// TIA Portal V20 export
ORGANIZATION_BLOCK "Main"   // OB1, LAD, ProgramCycle
TITLE = "Main Program Sweep (Cycle)"
{ S7_Optimized_Access := 'TRUE' }
// stored: SetENOAutomatically false
   VAR_INPUT
      Initial_Call : Bool;   // Initial call of this OB
      Remanence : Bool;   // =True, if remanent data are available
   END_VAR
BEGIN

REGION Network 1
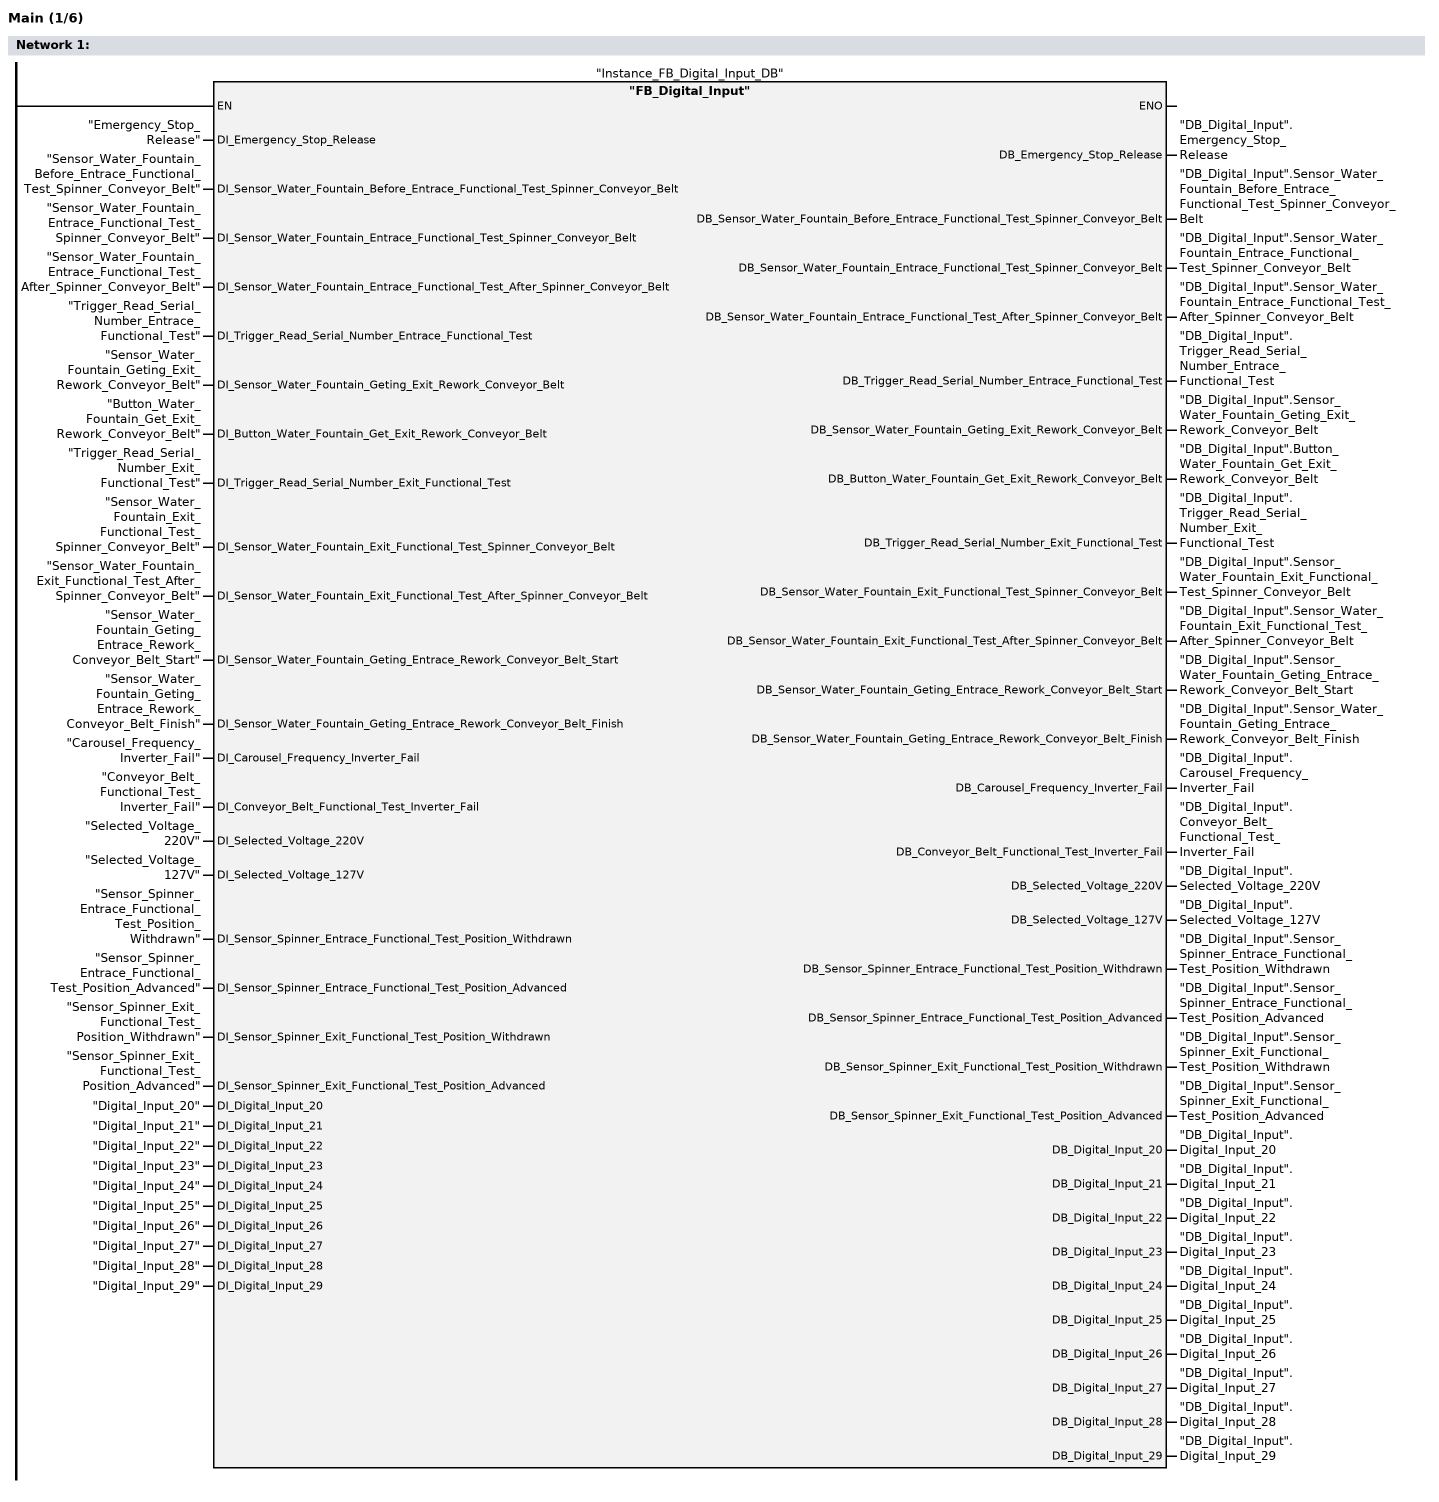
   RUNG wire#powerrail
      "Instance_FB_Digital_Input_DB"(DI_Emergency_Stop_Release := "Emergency_Stop_Release", DI_Sensor_Water_Fountain_Before_Entrace_Functional_Test_Spinner_Conveyor_Belt := "Sensor_Water_Fountain_Before_Entrace_Functional_Test_Spinner_Conveyor_Belt", DI_Sensor_Water_Fountain_Entrace_Functional_Test_Spinner_Conveyor_Belt := "Sensor_Water_Fountain_Entrace_Functional_Test_Spinner_Conveyor_Belt", DI_Sensor_Water_Fountain_Entrace_Functional_Test_After_Spinner_Conveyor_Belt := "Sensor_Water_Fountain_Entrace_Functional_Test_After_Spinner_Conveyor_Belt", DI_Trigger_Read_Serial_Number_Entrace_Functional_Test := "Trigger_Read_Serial_Number_Entrace_Functional_Test", DI_Sensor_Water_Fountain_Geting_Exit_Rework_Conveyor_Belt := "Sensor_Water_Fountain_Geting_Exit_Rework_Conveyor_Belt", DI_Button_Water_Fountain_Get_Exit_Rework_Conveyor_Belt := "Button_Water_Fountain_Get_Exit_Rework_Conveyor_Belt", DI_Trigger_Read_Serial_Number_Exit_Functional_Test := "Trigger_Read_Serial_Number_Exit_Functional_Test", DI_Sensor_Water_Fountain_Exit_Functional_Test_Spinner_Conveyor_Belt := "Sensor_Water_Fountain_Exit_Functional_Test_Spinner_Conveyor_Belt", DI_Sensor_Water_Fountain_Exit_Functional_Test_After_Spinner_Conveyor_Belt := "Sensor_Water_Fountain_Exit_Functional_Test_After_Spinner_Conveyor_Belt", DI_Sensor_Water_Fountain_Geting_Entrace_Rework_Conveyor_Belt_Start := "Sensor_Water_Fountain_Geting_Entrace_Rework_Conveyor_Belt_Start", DI_Sensor_Water_Fountain_Geting_Entrace_Rework_Conveyor_Belt_Finish := "Sensor_Water_Fountain_Geting_Entrace_Rework_Conveyor_Belt_Finish", DI_Carousel_Frequency_Inverter_Fail := "Carousel_Frequency_Inverter_Fail", DI_Conveyor_Belt_Functional_Test_Inverter_Fail := "Conveyor_Belt_Functional_Test_Inverter_Fail", DI_Selected_Voltage_220V := "Selected_Voltage_220V", DI_Selected_Voltage_127V := "Selected_Voltage_127V", DI_Sensor_Spinner_Entrace_Functional_Test_Position_Withdrawn := "Sensor_Spinner_Entrace_Functional_Test_Position_Withdrawn", DI_Sensor_Spinner_Entrace_Functional_Test_Position_Advanced := "Sensor_Spinner_Entrace_Functional_Test_Position_Advanced", DI_Sensor_Spinner_Exit_Functional_Test_Position_Withdrawn := "Sensor_Spinner_Exit_Functional_Test_Position_Withdrawn", DI_Sensor_Spinner_Exit_Functional_Test_Position_Advanced := "Sensor_Spinner_Exit_Functional_Test_Position_Advanced", DI_Digital_Input_20 := "Digital_Input_20", DI_Digital_Input_21 := "Digital_Input_21", DI_Digital_Input_22 := "Digital_Input_22", DI_Digital_Input_23 := "Digital_Input_23", DI_Digital_Input_24 := "Digital_Input_24", DI_Digital_Input_25 := "Digital_Input_25", DI_Digital_Input_26 := "Digital_Input_26", DI_Digital_Input_27 := "Digital_Input_27", DI_Digital_Input_28 := "Digital_Input_28", DI_Digital_Input_29 := "Digital_Input_29", DB_Emergency_Stop_Release => "DB_Digital_Input".Emergency_Stop_Release, DB_Sensor_Water_Fountain_Before_Entrace_Functional_Test_Spinner_Conveyor_Belt => "DB_Digital_Input".Sensor_Water_Fountain_Before_Entrace_Functional_Test_Spinner_Conveyor_Belt, DB_Sensor_Water_Fountain_Entrace_Functional_Test_Spinner_Conveyor_Belt => "DB_Digital_Input".Sensor_Water_Fountain_Entrace_Functional_Test_Spinner_Conveyor_Belt, DB_Sensor_Water_Fountain_Entrace_Functional_Test_After_Spinner_Conveyor_Belt => "DB_Digital_Input".Sensor_Water_Fountain_Entrace_Functional_Test_After_Spinner_Conveyor_Belt, DB_Trigger_Read_Serial_Number_Entrace_Functional_Test => "DB_Digital_Input".Trigger_Read_Serial_Number_Entrace_Functional_Test, DB_Sensor_Water_Fountain_Geting_Exit_Rework_Conveyor_Belt => "DB_Digital_Input".Sensor_Water_Fountain_Geting_Exit_Rework_Conveyor_Belt, DB_Button_Water_Fountain_Get_Exit_Rework_Conveyor_Belt => "DB_Digital_Input".Button_Water_Fountain_Get_Exit_Rework_Conveyor_Belt, DB_Trigger_Read_Serial_Number_Exit_Functional_Test => "DB_Digital_Input".Trigger_Read_Serial_Number_Exit_Functional_Test, DB_Sensor_Water_Fountain_Exit_Functional_Test_Spinner_Conveyor_Belt => "DB_Digital_Input".Sensor_Water_Fountain_Exit_Functional_Test_Spinner_Conveyor_Belt, DB_Sensor_Water_Fountain_Exit_Functional_Test_After_Spinner_Conveyor_Belt => "DB_Digital_Input".Sensor_Water_Fountain_Exit_Functional_Test_After_Spinner_Conveyor_Belt, DB_Sensor_Water_Fountain_Geting_Entrace_Rework_Conveyor_Belt_Start => "DB_Digital_Input".Sensor_Water_Fountain_Geting_Entrace_Rework_Conveyor_Belt_Start, DB_Sensor_Water_Fountain_Geting_Entrace_Rework_Conveyor_Belt_Finish => "DB_Digital_Input".Sensor_Water_Fountain_Geting_Entrace_Rework_Conveyor_Belt_Finish, DB_Carousel_Frequency_Inverter_Fail => "DB_Digital_Input".Carousel_Frequency_Inverter_Fail, DB_Conveyor_Belt_Functional_Test_Inverter_Fail => "DB_Digital_Input".Conveyor_Belt_Functional_Test_Inverter_Fail, DB_Selected_Voltage_220V => "DB_Digital_Input".Selected_Voltage_220V, DB_Selected_Voltage_127V => "DB_Digital_Input".Selected_Voltage_127V, DB_Sensor_Spinner_Entrace_Functional_Test_Position_Withdrawn => "DB_Digital_Input".Sensor_Spinner_Entrace_Functional_Test_Position_Withdrawn, DB_Sensor_Spinner_Entrace_Functional_Test_Position_Advanced => "DB_Digital_Input".Sensor_Spinner_Entrace_Functional_Test_Position_Advanced, DB_Sensor_Spinner_Exit_Functional_Test_Position_Withdrawn => "DB_Digital_Input".Sensor_Spinner_Exit_Functional_Test_Position_Withdrawn, DB_Sensor_Spinner_Exit_Functional_Test_Position_Advanced => "DB_Digital_Input".Sensor_Spinner_Exit_Functional_Test_Position_Advanced, DB_Digital_Input_20 => "DB_Digital_Input".Digital_Input_20, DB_Digital_Input_21 => "DB_Digital_Input".Digital_Input_21, DB_Digital_Input_22 => "DB_Digital_Input".Digital_Input_22, DB_Digital_Input_23 => "DB_Digital_Input".Digital_Input_23, DB_Digital_Input_24 => "DB_Digital_Input".Digital_Input_24, DB_Digital_Input_25 => "DB_Digital_Input".Digital_Input_25, DB_Digital_Input_26 => "DB_Digital_Input".Digital_Input_26, DB_Digital_Input_27 => "DB_Digital_Input".Digital_Input_27, DB_Digital_Input_28 => "DB_Digital_Input".Digital_Input_28, DB_Digital_Input_29 => "DB_Digital_Input".Digital_Input_29)
   END_RUNG
   // the same network as SCL:
   "Instance_FB_Digital_Input_DB"(DI_Emergency_Stop_Release := "Emergency_Stop_Release",   // "FB_Digital_Input"
                           DI_Sensor_Water_Fountain_Before_Entrace_Functional_Test_Spinner_Conveyor_Belt := "Sensor_Water_Fountain_Before_Entrace_Functional_Test_Spinner_Conveyor_Belt",
                           DI_Sensor_Water_Fountain_Entrace_Functional_Test_Spinner_Conveyor_Belt := "Sensor_Water_Fountain_Entrace_Functional_Test_Spinner_Conveyor_Belt",
                           DI_Sensor_Water_Fountain_Entrace_Functional_Test_After_Spinner_Conveyor_Belt := "Sensor_Water_Fountain_Entrace_Functional_Test_After_Spinner_Conveyor_Belt",
                           DI_Trigger_Read_Serial_Number_Entrace_Functional_Test := "Trigger_Read_Serial_Number_Entrace_Functional_Test",
                           DI_Sensor_Water_Fountain_Geting_Exit_Rework_Conveyor_Belt := "Sensor_Water_Fountain_Geting_Exit_Rework_Conveyor_Belt",
                           DI_Button_Water_Fountain_Get_Exit_Rework_Conveyor_Belt := "Button_Water_Fountain_Get_Exit_Rework_Conveyor_Belt",
                           DI_Trigger_Read_Serial_Number_Exit_Functional_Test := "Trigger_Read_Serial_Number_Exit_Functional_Test",
                           DI_Sensor_Water_Fountain_Exit_Functional_Test_Spinner_Conveyor_Belt := "Sensor_Water_Fountain_Exit_Functional_Test_Spinner_Conveyor_Belt",
                           DI_Sensor_Water_Fountain_Exit_Functional_Test_After_Spinner_Conveyor_Belt := "Sensor_Water_Fountain_Exit_Functional_Test_After_Spinner_Conveyor_Belt",
                           DI_Sensor_Water_Fountain_Geting_Entrace_Rework_Conveyor_Belt_Start := "Sensor_Water_Fountain_Geting_Entrace_Rework_Conveyor_Belt_Start",
                           DI_Sensor_Water_Fountain_Geting_Entrace_Rework_Conveyor_Belt_Finish := "Sensor_Water_Fountain_Geting_Entrace_Rework_Conveyor_Belt_Finish",
                           DI_Carousel_Frequency_Inverter_Fail := "Carousel_Frequency_Inverter_Fail",
                           DI_Conveyor_Belt_Functional_Test_Inverter_Fail := "Conveyor_Belt_Functional_Test_Inverter_Fail",
                           DI_Selected_Voltage_220V := "Selected_Voltage_220V",
                           DI_Selected_Voltage_127V := "Selected_Voltage_127V",
                           DI_Sensor_Spinner_Entrace_Functional_Test_Position_Withdrawn := "Sensor_Spinner_Entrace_Functional_Test_Position_Withdrawn",
                           DI_Sensor_Spinner_Entrace_Functional_Test_Position_Advanced := "Sensor_Spinner_Entrace_Functional_Test_Position_Advanced",
                           DI_Sensor_Spinner_Exit_Functional_Test_Position_Withdrawn := "Sensor_Spinner_Exit_Functional_Test_Position_Withdrawn",
                           DI_Sensor_Spinner_Exit_Functional_Test_Position_Advanced := "Sensor_Spinner_Exit_Functional_Test_Position_Advanced",
                           DI_Digital_Input_20 := "Digital_Input_20",
                           DI_Digital_Input_21 := "Digital_Input_21",
                           DI_Digital_Input_22 := "Digital_Input_22",
                           DI_Digital_Input_23 := "Digital_Input_23",
                           DI_Digital_Input_24 := "Digital_Input_24",
                           DI_Digital_Input_25 := "Digital_Input_25",
                           DI_Digital_Input_26 := "Digital_Input_26",
                           DI_Digital_Input_27 := "Digital_Input_27",
                           DI_Digital_Input_28 := "Digital_Input_28",
                           DI_Digital_Input_29 := "Digital_Input_29",
                           DB_Emergency_Stop_Release => "DB_Digital_Input".Emergency_Stop_Release,
                           DB_Sensor_Water_Fountain_Before_Entrace_Functional_Test_Spinner_Conveyor_Belt => "DB_Digital_Input".Sensor_Water_Fountain_Before_Entrace_Functional_Test_Spinner_Conveyor_Belt,
                           DB_Sensor_Water_Fountain_Entrace_Functional_Test_Spinner_Conveyor_Belt => "DB_Digital_Input".Sensor_Water_Fountain_Entrace_Functional_Test_Spinner_Conveyor_Belt,
                           DB_Sensor_Water_Fountain_Entrace_Functional_Test_After_Spinner_Conveyor_Belt => "DB_Digital_Input".Sensor_Water_Fountain_Entrace_Functional_Test_After_Spinner_Conveyor_Belt,
                           DB_Trigger_Read_Serial_Number_Entrace_Functional_Test => "DB_Digital_Input".Trigger_Read_Serial_Number_Entrace_Functional_Test,
                           DB_Sensor_Water_Fountain_Geting_Exit_Rework_Conveyor_Belt => "DB_Digital_Input".Sensor_Water_Fountain_Geting_Exit_Rework_Conveyor_Belt,
                           DB_Button_Water_Fountain_Get_Exit_Rework_Conveyor_Belt => "DB_Digital_Input".Button_Water_Fountain_Get_Exit_Rework_Conveyor_Belt,
                           DB_Trigger_Read_Serial_Number_Exit_Functional_Test => "DB_Digital_Input".Trigger_Read_Serial_Number_Exit_Functional_Test,
                           DB_Sensor_Water_Fountain_Exit_Functional_Test_Spinner_Conveyor_Belt => "DB_Digital_Input".Sensor_Water_Fountain_Exit_Functional_Test_Spinner_Conveyor_Belt,
                           DB_Sensor_Water_Fountain_Exit_Functional_Test_After_Spinner_Conveyor_Belt => "DB_Digital_Input".Sensor_Water_Fountain_Exit_Functional_Test_After_Spinner_Conveyor_Belt,
                           DB_Sensor_Water_Fountain_Geting_Entrace_Rework_Conveyor_Belt_Start => "DB_Digital_Input".Sensor_Water_Fountain_Geting_Entrace_Rework_Conveyor_Belt_Start,
                           DB_Sensor_Water_Fountain_Geting_Entrace_Rework_Conveyor_Belt_Finish => "DB_Digital_Input".Sensor_Water_Fountain_Geting_Entrace_Rework_Conveyor_Belt_Finish,
                           DB_Carousel_Frequency_Inverter_Fail => "DB_Digital_Input".Carousel_Frequency_Inverter_Fail,
                           DB_Conveyor_Belt_Functional_Test_Inverter_Fail => "DB_Digital_Input".Conveyor_Belt_Functional_Test_Inverter_Fail,
                           DB_Selected_Voltage_220V => "DB_Digital_Input".Selected_Voltage_220V,
                           DB_Selected_Voltage_127V => "DB_Digital_Input".Selected_Voltage_127V,
                           DB_Sensor_Spinner_Entrace_Functional_Test_Position_Withdrawn => "DB_Digital_Input".Sensor_Spinner_Entrace_Functional_Test_Position_Withdrawn,
                           DB_Sensor_Spinner_Entrace_Functional_Test_Position_Advanced => "DB_Digital_Input".Sensor_Spinner_Entrace_Functional_Test_Position_Advanced,
                           DB_Sensor_Spinner_Exit_Functional_Test_Position_Withdrawn => "DB_Digital_Input".Sensor_Spinner_Exit_Functional_Test_Position_Withdrawn,
                           DB_Sensor_Spinner_Exit_Functional_Test_Position_Advanced => "DB_Digital_Input".Sensor_Spinner_Exit_Functional_Test_Position_Advanced,
                           DB_Digital_Input_20 => "DB_Digital_Input".Digital_Input_20,
                           DB_Digital_Input_21 => "DB_Digital_Input".Digital_Input_21,
                           DB_Digital_Input_22 => "DB_Digital_Input".Digital_Input_22,
                           DB_Digital_Input_23 => "DB_Digital_Input".Digital_Input_23,
                           DB_Digital_Input_24 => "DB_Digital_Input".Digital_Input_24,
                           DB_Digital_Input_25 => "DB_Digital_Input".Digital_Input_25,
                           DB_Digital_Input_26 => "DB_Digital_Input".Digital_Input_26,
                           DB_Digital_Input_27 => "DB_Digital_Input".Digital_Input_27,
                           DB_Digital_Input_28 => "DB_Digital_Input".Digital_Input_28,
                           DB_Digital_Input_29 => "DB_Digital_Input".Digital_Input_29);
END_REGION

REGION Network 2
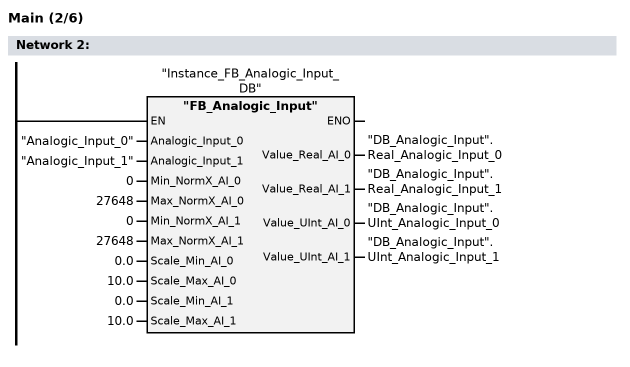
   RUNG wire#powerrail
      "Instance_FB_Analogic_Input_DB"(Analogic_Input_0 := "Analogic_Input_0", Analogic_Input_1 := "Analogic_Input_1", Min_NormX_AI_0 := 0, Max_NormX_AI_0 := 27648, Min_NormX_AI_1 := 0, Max_NormX_AI_1 := 27648, Scale_Min_AI_0 := 0.0, Scale_Max_AI_0 := 10.0, Scale_Min_AI_1 := 0.0, Scale_Max_AI_1 := 10.0, Value_Real_AI_0 => "DB_Analogic_Input".Real_Analogic_Input_0, Value_Real_AI_1 => "DB_Analogic_Input".Real_Analogic_Input_1, Value_UInt_AI_0 => "DB_Analogic_Input".UInt_Analogic_Input_0, Value_UInt_AI_1 => "DB_Analogic_Input".UInt_Analogic_Input_1)
   END_RUNG
   // the same network as SCL:
   "Instance_FB_Analogic_Input_DB"(Analogic_Input_0 := "Analogic_Input_0",   // "FB_Analogic_Input"
                           Analogic_Input_1 := "Analogic_Input_1",
                           Min_NormX_AI_0 := 0,
                           Max_NormX_AI_0 := 27648,
                           Min_NormX_AI_1 := 0,
                           Max_NormX_AI_1 := 27648,
                           Scale_Min_AI_0 := 0.0,
                           Scale_Max_AI_0 := 10.0,
                           Scale_Min_AI_1 := 0.0,
                           Scale_Max_AI_1 := 10.0,
                           Value_Real_AI_0 => "DB_Analogic_Input".Real_Analogic_Input_0,
                           Value_Real_AI_1 => "DB_Analogic_Input".Real_Analogic_Input_1,
                           Value_UInt_AI_0 => "DB_Analogic_Input".UInt_Analogic_Input_0,
                           Value_UInt_AI_1 => "DB_Analogic_Input".UInt_Analogic_Input_1);
END_REGION

REGION Network 3
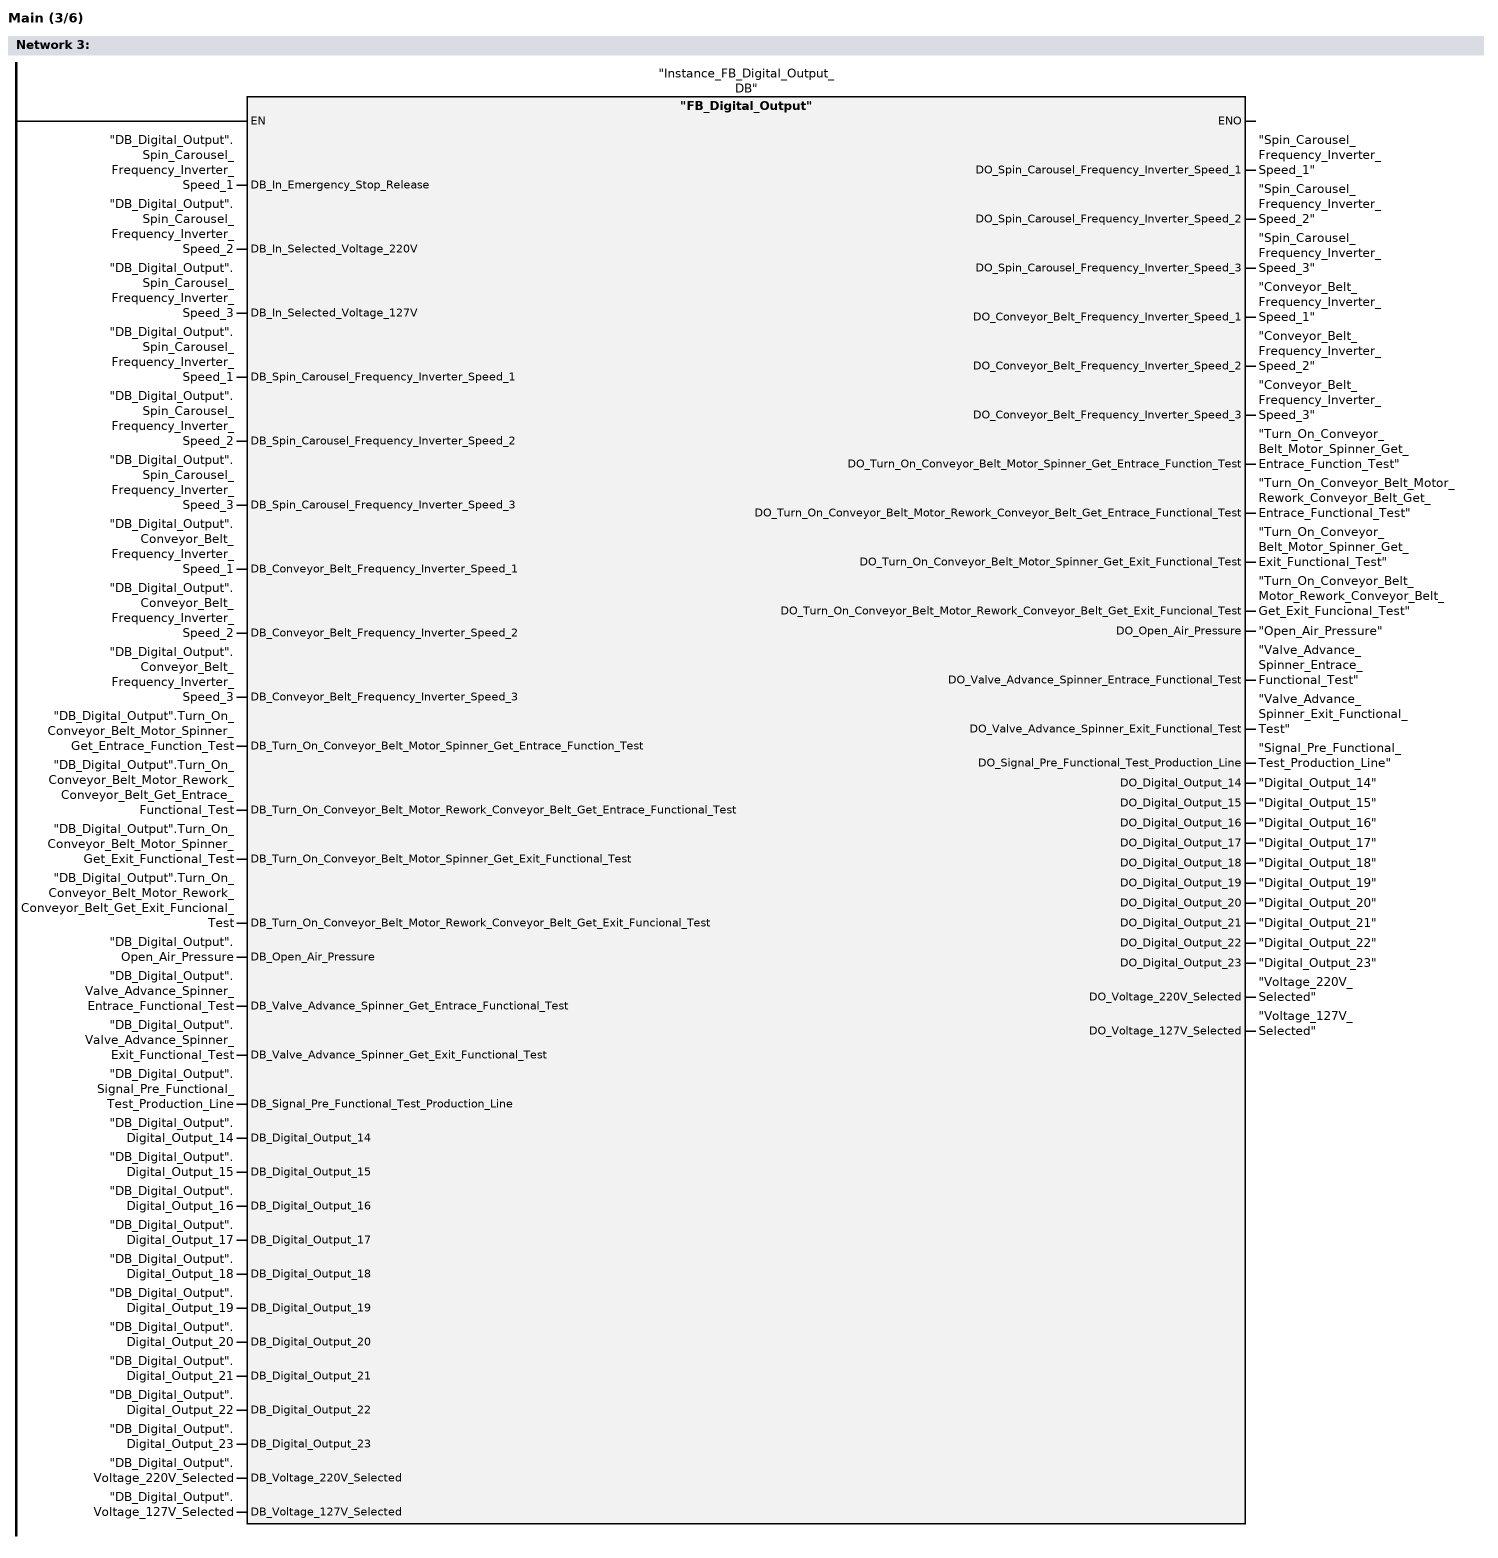
   RUNG wire#powerrail
      "Instance_FB_Digital_Output_DB"(DB_In_Emergency_Stop_Release := "DB_Digital_Output".Spin_Carousel_Frequency_Inverter_Speed_1, DB_In_Selected_Voltage_220V := "DB_Digital_Output".Spin_Carousel_Frequency_Inverter_Speed_2, DB_In_Selected_Voltage_127V := "DB_Digital_Output".Spin_Carousel_Frequency_Inverter_Speed_3, DB_Spin_Carousel_Frequency_Inverter_Speed_1 := "DB_Digital_Output".Spin_Carousel_Frequency_Inverter_Speed_1, DB_Spin_Carousel_Frequency_Inverter_Speed_2 := "DB_Digital_Output".Spin_Carousel_Frequency_Inverter_Speed_2, DB_Spin_Carousel_Frequency_Inverter_Speed_3 := "DB_Digital_Output".Spin_Carousel_Frequency_Inverter_Speed_3, DB_Conveyor_Belt_Frequency_Inverter_Speed_1 := "DB_Digital_Output".Conveyor_Belt_Frequency_Inverter_Speed_1, DB_Conveyor_Belt_Frequency_Inverter_Speed_2 := "DB_Digital_Output".Conveyor_Belt_Frequency_Inverter_Speed_2, DB_Conveyor_Belt_Frequency_Inverter_Speed_3 := "DB_Digital_Output".Conveyor_Belt_Frequency_Inverter_Speed_3, DB_Turn_On_Conveyor_Belt_Motor_Spinner_Get_Entrace_Function_Test := "DB_Digital_Output".Turn_On_Conveyor_Belt_Motor_Spinner_Get_Entrace_Function_Test, DB_Turn_On_Conveyor_Belt_Motor_Rework_Conveyor_Belt_Get_Entrace_Functional_Test := "DB_Digital_Output".Turn_On_Conveyor_Belt_Motor_Rework_Conveyor_Belt_Get_Entrace_Functional_Test, DB_Turn_On_Conveyor_Belt_Motor_Spinner_Get_Exit_Functional_Test := "DB_Digital_Output".Turn_On_Conveyor_Belt_Motor_Spinner_Get_Exit_Functional_Test, DB_Turn_On_Conveyor_Belt_Motor_Rework_Conveyor_Belt_Get_Exit_Funcional_Test := "DB_Digital_Output".Turn_On_Conveyor_Belt_Motor_Rework_Conveyor_Belt_Get_Exit_Funcional_Test, DB_Open_Air_Pressure := "DB_Digital_Output".Open_Air_Pressure, DB_Valve_Advance_Spinner_Get_Entrace_Functional_Test := "DB_Digital_Output".Valve_Advance_Spinner_Entrace_Functional_Test, DB_Valve_Advance_Spinner_Get_Exit_Functional_Test := "DB_Digital_Output".Valve_Advance_Spinner_Exit_Functional_Test, DB_Signal_Pre_Functional_Test_Production_Line := "DB_Digital_Output".Signal_Pre_Functional_Test_Production_Line, DB_Digital_Output_14 := "DB_Digital_Output".Digital_Output_14, DB_Digital_Output_15 := "DB_Digital_Output".Digital_Output_15, DB_Digital_Output_16 := "DB_Digital_Output".Digital_Output_16, DB_Digital_Output_17 := "DB_Digital_Output".Digital_Output_17, DB_Digital_Output_18 := "DB_Digital_Output".Digital_Output_18, DB_Digital_Output_19 := "DB_Digital_Output".Digital_Output_19, DB_Digital_Output_20 := "DB_Digital_Output".Digital_Output_20, DB_Digital_Output_21 := "DB_Digital_Output".Digital_Output_21, DB_Digital_Output_22 := "DB_Digital_Output".Digital_Output_22, DB_Digital_Output_23 := "DB_Digital_Output".Digital_Output_23, DB_Voltage_220V_Selected := "DB_Digital_Output".Voltage_220V_Selected, DB_Voltage_127V_Selected := "DB_Digital_Output".Voltage_127V_Selected, DO_Spin_Carousel_Frequency_Inverter_Speed_1 => "Spin_Carousel_Frequency_Inverter_Speed_1", DO_Spin_Carousel_Frequency_Inverter_Speed_2 => "Spin_Carousel_Frequency_Inverter_Speed_2", DO_Spin_Carousel_Frequency_Inverter_Speed_3 => "Spin_Carousel_Frequency_Inverter_Speed_3", DO_Conveyor_Belt_Frequency_Inverter_Speed_1 => "Conveyor_Belt_Frequency_Inverter_Speed_1", DO_Conveyor_Belt_Frequency_Inverter_Speed_2 => "Conveyor_Belt_Frequency_Inverter_Speed_2", DO_Conveyor_Belt_Frequency_Inverter_Speed_3 => "Conveyor_Belt_Frequency_Inverter_Speed_3", DO_Turn_On_Conveyor_Belt_Motor_Spinner_Get_Entrace_Function_Test => "Turn_On_Conveyor_Belt_Motor_Spinner_Get_Entrace_Function_Test", DO_Turn_On_Conveyor_Belt_Motor_Rework_Conveyor_Belt_Get_Entrace_Functional_Test => "Turn_On_Conveyor_Belt_Motor_Rework_Conveyor_Belt_Get_Entrace_Functional_Test", DO_Turn_On_Conveyor_Belt_Motor_Spinner_Get_Exit_Functional_Test => "Turn_On_Conveyor_Belt_Motor_Spinner_Get_Exit_Functional_Test", DO_Turn_On_Conveyor_Belt_Motor_Rework_Conveyor_Belt_Get_Exit_Funcional_Test => "Turn_On_Conveyor_Belt_Motor_Rework_Conveyor_Belt_Get_Exit_Funcional_Test", DO_Open_Air_Pressure => "Open_Air_Pressure", DO_Valve_Advance_Spinner_Entrace_Functional_Test => "Valve_Advance_Spinner_Entrace_Functional_Test", DO_Valve_Advance_Spinner_Exit_Functional_Test => "Valve_Advance_Spinner_Exit_Functional_Test", DO_Signal_Pre_Functional_Test_Production_Line => "Signal_Pre_Functional_Test_Production_Line", DO_Digital_Output_14 => "Digital_Output_14", DO_Digital_Output_15 => "Digital_Output_15", DO_Digital_Output_16 => "Digital_Output_16", DO_Digital_Output_17 => "Digital_Output_17", DO_Digital_Output_18 => "Digital_Output_18", DO_Digital_Output_19 => "Digital_Output_19", DO_Digital_Output_20 => "Digital_Output_20", DO_Digital_Output_21 => "Digital_Output_21", DO_Digital_Output_22 => "Digital_Output_22", DO_Digital_Output_23 => "Digital_Output_23", DO_Voltage_220V_Selected => "Voltage_220V_Selected", DO_Voltage_127V_Selected => "Voltage_127V_Selected")
   END_RUNG
   // the same network as SCL:
   "Instance_FB_Digital_Output_DB"(DB_In_Emergency_Stop_Release := "DB_Digital_Output".Spin_Carousel_Frequency_Inverter_Speed_1,   // "FB_Digital_Output"
                           DB_In_Selected_Voltage_220V := "DB_Digital_Output".Spin_Carousel_Frequency_Inverter_Speed_2,
                           DB_In_Selected_Voltage_127V := "DB_Digital_Output".Spin_Carousel_Frequency_Inverter_Speed_3,
                           DB_Spin_Carousel_Frequency_Inverter_Speed_1 := "DB_Digital_Output".Spin_Carousel_Frequency_Inverter_Speed_1,
                           DB_Spin_Carousel_Frequency_Inverter_Speed_2 := "DB_Digital_Output".Spin_Carousel_Frequency_Inverter_Speed_2,
                           DB_Spin_Carousel_Frequency_Inverter_Speed_3 := "DB_Digital_Output".Spin_Carousel_Frequency_Inverter_Speed_3,
                           DB_Conveyor_Belt_Frequency_Inverter_Speed_1 := "DB_Digital_Output".Conveyor_Belt_Frequency_Inverter_Speed_1,
                           DB_Conveyor_Belt_Frequency_Inverter_Speed_2 := "DB_Digital_Output".Conveyor_Belt_Frequency_Inverter_Speed_2,
                           DB_Conveyor_Belt_Frequency_Inverter_Speed_3 := "DB_Digital_Output".Conveyor_Belt_Frequency_Inverter_Speed_3,
                           DB_Turn_On_Conveyor_Belt_Motor_Spinner_Get_Entrace_Function_Test := "DB_Digital_Output".Turn_On_Conveyor_Belt_Motor_Spinner_Get_Entrace_Function_Test,
                           DB_Turn_On_Conveyor_Belt_Motor_Rework_Conveyor_Belt_Get_Entrace_Functional_Test := "DB_Digital_Output".Turn_On_Conveyor_Belt_Motor_Rework_Conveyor_Belt_Get_Entrace_Functional_Test,
                           DB_Turn_On_Conveyor_Belt_Motor_Spinner_Get_Exit_Functional_Test := "DB_Digital_Output".Turn_On_Conveyor_Belt_Motor_Spinner_Get_Exit_Functional_Test,
                           DB_Turn_On_Conveyor_Belt_Motor_Rework_Conveyor_Belt_Get_Exit_Funcional_Test := "DB_Digital_Output".Turn_On_Conveyor_Belt_Motor_Rework_Conveyor_Belt_Get_Exit_Funcional_Test,
                           DB_Open_Air_Pressure := "DB_Digital_Output".Open_Air_Pressure,
                           DB_Valve_Advance_Spinner_Get_Entrace_Functional_Test := "DB_Digital_Output".Valve_Advance_Spinner_Entrace_Functional_Test,
                           DB_Valve_Advance_Spinner_Get_Exit_Functional_Test := "DB_Digital_Output".Valve_Advance_Spinner_Exit_Functional_Test,
                           DB_Signal_Pre_Functional_Test_Production_Line := "DB_Digital_Output".Signal_Pre_Functional_Test_Production_Line,
                           DB_Digital_Output_14 := "DB_Digital_Output".Digital_Output_14,
                           DB_Digital_Output_15 := "DB_Digital_Output".Digital_Output_15,
                           DB_Digital_Output_16 := "DB_Digital_Output".Digital_Output_16,
                           DB_Digital_Output_17 := "DB_Digital_Output".Digital_Output_17,
                           DB_Digital_Output_18 := "DB_Digital_Output".Digital_Output_18,
                           DB_Digital_Output_19 := "DB_Digital_Output".Digital_Output_19,
                           DB_Digital_Output_20 := "DB_Digital_Output".Digital_Output_20,
                           DB_Digital_Output_21 := "DB_Digital_Output".Digital_Output_21,
                           DB_Digital_Output_22 := "DB_Digital_Output".Digital_Output_22,
                           DB_Digital_Output_23 := "DB_Digital_Output".Digital_Output_23,
                           DB_Voltage_220V_Selected := "DB_Digital_Output".Voltage_220V_Selected,
                           DB_Voltage_127V_Selected := "DB_Digital_Output".Voltage_127V_Selected,
                           DO_Spin_Carousel_Frequency_Inverter_Speed_1 => "Spin_Carousel_Frequency_Inverter_Speed_1",
                           DO_Spin_Carousel_Frequency_Inverter_Speed_2 => "Spin_Carousel_Frequency_Inverter_Speed_2",
                           DO_Spin_Carousel_Frequency_Inverter_Speed_3 => "Spin_Carousel_Frequency_Inverter_Speed_3",
                           DO_Conveyor_Belt_Frequency_Inverter_Speed_1 => "Conveyor_Belt_Frequency_Inverter_Speed_1",
                           DO_Conveyor_Belt_Frequency_Inverter_Speed_2 => "Conveyor_Belt_Frequency_Inverter_Speed_2",
                           DO_Conveyor_Belt_Frequency_Inverter_Speed_3 => "Conveyor_Belt_Frequency_Inverter_Speed_3",
                           DO_Turn_On_Conveyor_Belt_Motor_Spinner_Get_Entrace_Function_Test => "Turn_On_Conveyor_Belt_Motor_Spinner_Get_Entrace_Function_Test",
                           DO_Turn_On_Conveyor_Belt_Motor_Rework_Conveyor_Belt_Get_Entrace_Functional_Test => "Turn_On_Conveyor_Belt_Motor_Rework_Conveyor_Belt_Get_Entrace_Functional_Test",
                           DO_Turn_On_Conveyor_Belt_Motor_Spinner_Get_Exit_Functional_Test => "Turn_On_Conveyor_Belt_Motor_Spinner_Get_Exit_Functional_Test",
                           DO_Turn_On_Conveyor_Belt_Motor_Rework_Conveyor_Belt_Get_Exit_Funcional_Test => "Turn_On_Conveyor_Belt_Motor_Rework_Conveyor_Belt_Get_Exit_Funcional_Test",
                           DO_Open_Air_Pressure => "Open_Air_Pressure",
                           DO_Valve_Advance_Spinner_Entrace_Functional_Test => "Valve_Advance_Spinner_Entrace_Functional_Test",
                           DO_Valve_Advance_Spinner_Exit_Functional_Test => "Valve_Advance_Spinner_Exit_Functional_Test",
                           DO_Signal_Pre_Functional_Test_Production_Line => "Signal_Pre_Functional_Test_Production_Line",
                           DO_Digital_Output_14 => "Digital_Output_14",
                           DO_Digital_Output_15 => "Digital_Output_15",
                           DO_Digital_Output_16 => "Digital_Output_16",
                           DO_Digital_Output_17 => "Digital_Output_17",
                           DO_Digital_Output_18 => "Digital_Output_18",
                           DO_Digital_Output_19 => "Digital_Output_19",
                           DO_Digital_Output_20 => "Digital_Output_20",
                           DO_Digital_Output_21 => "Digital_Output_21",
                           DO_Digital_Output_22 => "Digital_Output_22",
                           DO_Digital_Output_23 => "Digital_Output_23",
                           DO_Voltage_220V_Selected => "Voltage_220V_Selected",
                           DO_Voltage_127V_Selected => "Voltage_127V_Selected");
END_REGION

REGION Network 4
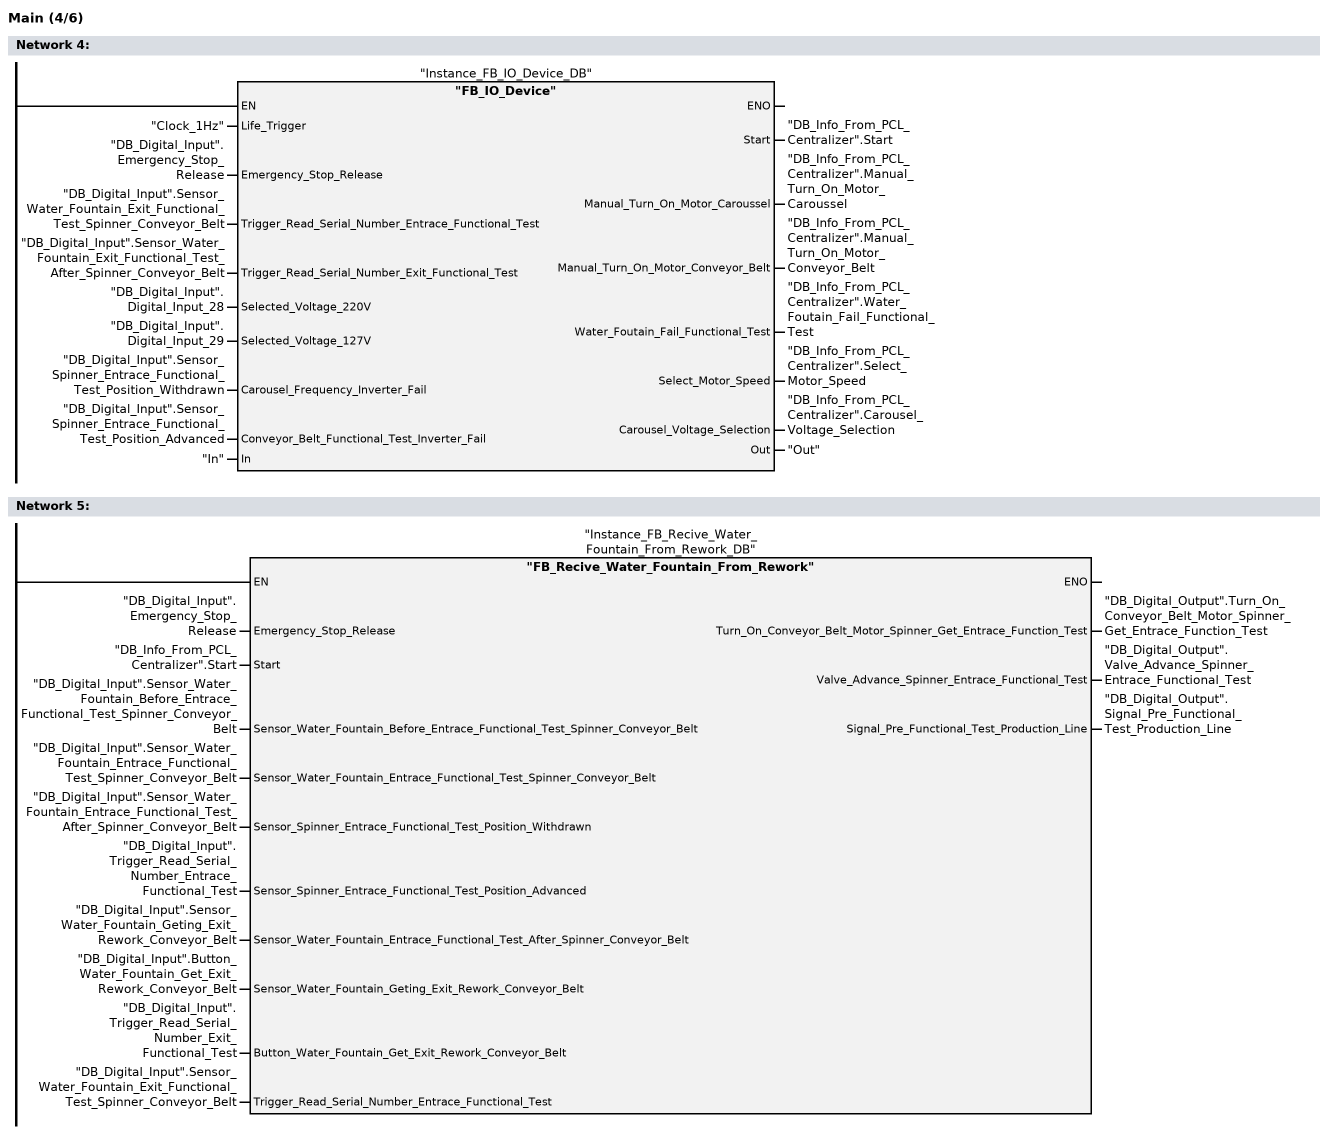
   RUNG wire#powerrail
      "Instance_FB_IO_Device_DB"(Life_Trigger := "Clock_1Hz", Emergency_Stop_Release := "DB_Digital_Input".Emergency_Stop_Release, Trigger_Read_Serial_Number_Entrace_Functional_Test := "DB_Digital_Input".Sensor_Water_Fountain_Exit_Functional_Test_Spinner_Conveyor_Belt, Trigger_Read_Serial_Number_Exit_Functional_Test := "DB_Digital_Input".Sensor_Water_Fountain_Exit_Functional_Test_After_Spinner_Conveyor_Belt, Selected_Voltage_220V := "DB_Digital_Input".Digital_Input_28, Selected_Voltage_127V := "DB_Digital_Input".Digital_Input_29, Carousel_Frequency_Inverter_Fail := "DB_Digital_Input".Sensor_Spinner_Entrace_Functional_Test_Position_Withdrawn, Conveyor_Belt_Functional_Test_Inverter_Fail := "DB_Digital_Input".Sensor_Spinner_Entrace_Functional_Test_Position_Advanced, In := "In", Start => "DB_Info_From_PCL_Centralizer".Start, Manual_Turn_On_Motor_Caroussel => "DB_Info_From_PCL_Centralizer".Manual_Turn_On_Motor_Caroussel, Manual_Turn_On_Motor_Conveyor_Belt => "DB_Info_From_PCL_Centralizer".Manual_Turn_On_Motor_Conveyor_Belt, Water_Foutain_Fail_Functional_Test => "DB_Info_From_PCL_Centralizer".Water_Foutain_Fail_Functional_Test, Select_Motor_Speed => "DB_Info_From_PCL_Centralizer".Select_Motor_Speed, Carousel_Voltage_Selection => "DB_Info_From_PCL_Centralizer".Carousel_Voltage_Selection, Out => "Out")
   END_RUNG
   // the same network as SCL:
   "Instance_FB_IO_Device_DB"(Life_Trigger := "Clock_1Hz",   // "FB_IO_Device"
                           Emergency_Stop_Release := "DB_Digital_Input".Emergency_Stop_Release,
                           Trigger_Read_Serial_Number_Entrace_Functional_Test := "DB_Digital_Input".Sensor_Water_Fountain_Exit_Functional_Test_Spinner_Conveyor_Belt,
                           Trigger_Read_Serial_Number_Exit_Functional_Test := "DB_Digital_Input".Sensor_Water_Fountain_Exit_Functional_Test_After_Spinner_Conveyor_Belt,
                           Selected_Voltage_220V := "DB_Digital_Input".Digital_Input_28,
                           Selected_Voltage_127V := "DB_Digital_Input".Digital_Input_29,
                           Carousel_Frequency_Inverter_Fail := "DB_Digital_Input".Sensor_Spinner_Entrace_Functional_Test_Position_Withdrawn,
                           Conveyor_Belt_Functional_Test_Inverter_Fail := "DB_Digital_Input".Sensor_Spinner_Entrace_Functional_Test_Position_Advanced,
                           In := "In",
                           Start => "DB_Info_From_PCL_Centralizer".Start,
                           Manual_Turn_On_Motor_Caroussel => "DB_Info_From_PCL_Centralizer".Manual_Turn_On_Motor_Caroussel,
                           Manual_Turn_On_Motor_Conveyor_Belt => "DB_Info_From_PCL_Centralizer".Manual_Turn_On_Motor_Conveyor_Belt,
                           Water_Foutain_Fail_Functional_Test => "DB_Info_From_PCL_Centralizer".Water_Foutain_Fail_Functional_Test,
                           Select_Motor_Speed => "DB_Info_From_PCL_Centralizer".Select_Motor_Speed,
                           Carousel_Voltage_Selection => "DB_Info_From_PCL_Centralizer".Carousel_Voltage_Selection,
                           Out => "Out");
END_REGION

REGION Network 5
   RUNG wire#powerrail
      "Instance_FB_Recive_Water_Fountain_From_Rework_DB"(Emergency_Stop_Release := "DB_Digital_Input".Emergency_Stop_Release, Start := "DB_Info_From_PCL_Centralizer".Start, Sensor_Water_Fountain_Before_Entrace_Functional_Test_Spinner_Conveyor_Belt := "DB_Digital_Input".Sensor_Water_Fountain_Before_Entrace_Functional_Test_Spinner_Conveyor_Belt, Sensor_Water_Fountain_Entrace_Functional_Test_Spinner_Conveyor_Belt := "DB_Digital_Input".Sensor_Water_Fountain_Entrace_Functional_Test_Spinner_Conveyor_Belt, Sensor_Spinner_Entrace_Functional_Test_Position_Withdrawn := "DB_Digital_Input".Sensor_Water_Fountain_Entrace_Functional_Test_After_Spinner_Conveyor_Belt, Sensor_Spinner_Entrace_Functional_Test_Position_Advanced := "DB_Digital_Input".Trigger_Read_Serial_Number_Entrace_Functional_Test, Sensor_Water_Fountain_Entrace_Functional_Test_After_Spinner_Conveyor_Belt := "DB_Digital_Input".Sensor_Water_Fountain_Geting_Exit_Rework_Conveyor_Belt, Sensor_Water_Fountain_Geting_Exit_Rework_Conveyor_Belt := "DB_Digital_Input".Button_Water_Fountain_Get_Exit_Rework_Conveyor_Belt, Button_Water_Fountain_Get_Exit_Rework_Conveyor_Belt := "DB_Digital_Input".Trigger_Read_Serial_Number_Exit_Functional_Test, Trigger_Read_Serial_Number_Entrace_Functional_Test := "DB_Digital_Input".Sensor_Water_Fountain_Exit_Functional_Test_Spinner_Conveyor_Belt, Turn_On_Conveyor_Belt_Motor_Spinner_Get_Entrace_Function_Test => "DB_Digital_Output".Turn_On_Conveyor_Belt_Motor_Spinner_Get_Entrace_Function_Test, Valve_Advance_Spinner_Entrace_Functional_Test => "DB_Digital_Output".Valve_Advance_Spinner_Entrace_Functional_Test, Signal_Pre_Functional_Test_Production_Line => "DB_Digital_Output".Signal_Pre_Functional_Test_Production_Line)
   END_RUNG
   // the same network as SCL:
   "Instance_FB_Recive_Water_Fountain_From_Rework_DB"(Emergency_Stop_Release := "DB_Digital_Input".Emergency_Stop_Release,   // "FB_Recive_Water_Fountain_From_Rework"
                           Start := "DB_Info_From_PCL_Centralizer".Start,
                           Sensor_Water_Fountain_Before_Entrace_Functional_Test_Spinner_Conveyor_Belt := "DB_Digital_Input".Sensor_Water_Fountain_Before_Entrace_Functional_Test_Spinner_Conveyor_Belt,
                           Sensor_Water_Fountain_Entrace_Functional_Test_Spinner_Conveyor_Belt := "DB_Digital_Input".Sensor_Water_Fountain_Entrace_Functional_Test_Spinner_Conveyor_Belt,
                           Sensor_Spinner_Entrace_Functional_Test_Position_Withdrawn := "DB_Digital_Input".Sensor_Water_Fountain_Entrace_Functional_Test_After_Spinner_Conveyor_Belt,
                           Sensor_Spinner_Entrace_Functional_Test_Position_Advanced := "DB_Digital_Input".Trigger_Read_Serial_Number_Entrace_Functional_Test,
                           Sensor_Water_Fountain_Entrace_Functional_Test_After_Spinner_Conveyor_Belt := "DB_Digital_Input".Sensor_Water_Fountain_Geting_Exit_Rework_Conveyor_Belt,
                           Sensor_Water_Fountain_Geting_Exit_Rework_Conveyor_Belt := "DB_Digital_Input".Button_Water_Fountain_Get_Exit_Rework_Conveyor_Belt,
                           Button_Water_Fountain_Get_Exit_Rework_Conveyor_Belt := "DB_Digital_Input".Trigger_Read_Serial_Number_Exit_Functional_Test,
                           Trigger_Read_Serial_Number_Entrace_Functional_Test := "DB_Digital_Input".Sensor_Water_Fountain_Exit_Functional_Test_Spinner_Conveyor_Belt,
                           Turn_On_Conveyor_Belt_Motor_Spinner_Get_Entrace_Function_Test => "DB_Digital_Output".Turn_On_Conveyor_Belt_Motor_Spinner_Get_Entrace_Function_Test,
                           Valve_Advance_Spinner_Entrace_Functional_Test => "DB_Digital_Output".Valve_Advance_Spinner_Entrace_Functional_Test,
                           Signal_Pre_Functional_Test_Production_Line => "DB_Digital_Output".Signal_Pre_Functional_Test_Production_Line);
END_REGION

REGION Network 6
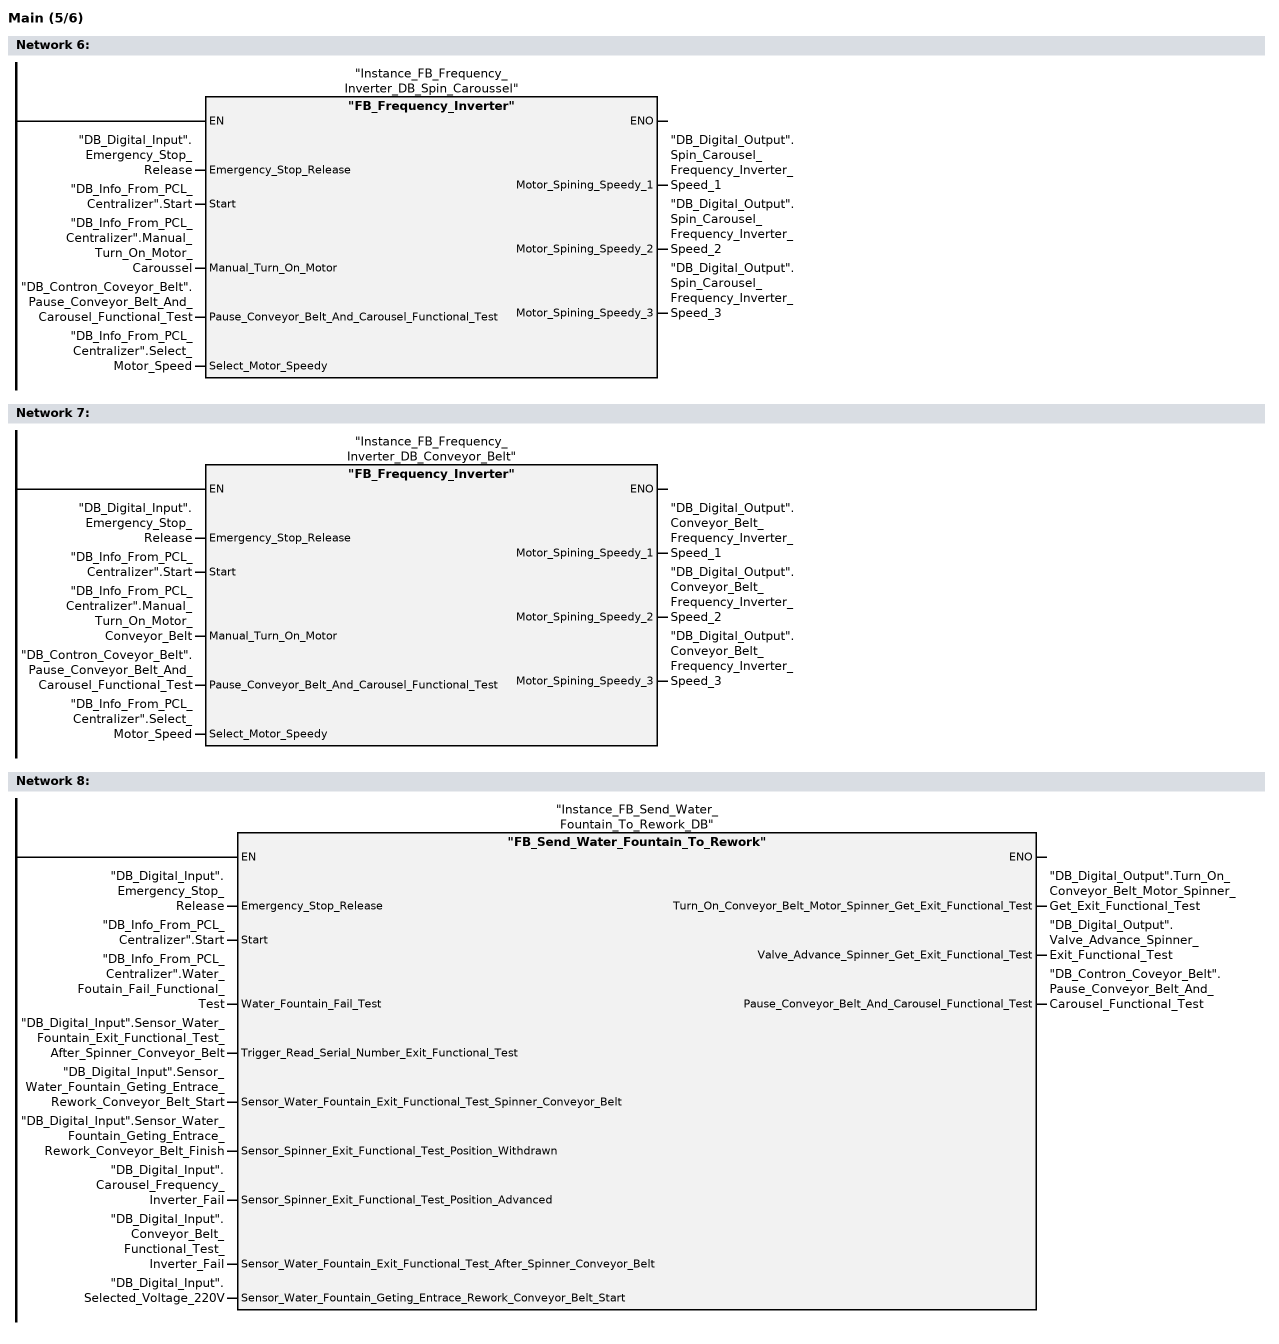
   RUNG wire#powerrail
      "Instance_FB_Frequency_Inverter_DB_Spin_Caroussel"(Emergency_Stop_Release := "DB_Digital_Input".Emergency_Stop_Release, Start := "DB_Info_From_PCL_Centralizer".Start, Manual_Turn_On_Motor := "DB_Info_From_PCL_Centralizer".Manual_Turn_On_Motor_Caroussel, Pause_Conveyor_Belt_And_Carousel_Functional_Test := "DB_Contron_Coveyor_Belt".Pause_Conveyor_Belt_And_Carousel_Functional_Test, Select_Motor_Speedy := "DB_Info_From_PCL_Centralizer".Select_Motor_Speed, Motor_Spining_Speedy_1 => "DB_Digital_Output".Spin_Carousel_Frequency_Inverter_Speed_1, Motor_Spining_Speedy_2 => "DB_Digital_Output".Spin_Carousel_Frequency_Inverter_Speed_2, Motor_Spining_Speedy_3 => "DB_Digital_Output".Spin_Carousel_Frequency_Inverter_Speed_3)
   END_RUNG
   // the same network as SCL:
   "Instance_FB_Frequency_Inverter_DB_Spin_Caroussel"(Emergency_Stop_Release := "DB_Digital_Input".Emergency_Stop_Release,   // "FB_Frequency_Inverter"
                           Start := "DB_Info_From_PCL_Centralizer".Start,
                           Manual_Turn_On_Motor := "DB_Info_From_PCL_Centralizer".Manual_Turn_On_Motor_Caroussel,
                           Pause_Conveyor_Belt_And_Carousel_Functional_Test := "DB_Contron_Coveyor_Belt".Pause_Conveyor_Belt_And_Carousel_Functional_Test,
                           Select_Motor_Speedy := "DB_Info_From_PCL_Centralizer".Select_Motor_Speed,
                           Motor_Spining_Speedy_1 => "DB_Digital_Output".Spin_Carousel_Frequency_Inverter_Speed_1,
                           Motor_Spining_Speedy_2 => "DB_Digital_Output".Spin_Carousel_Frequency_Inverter_Speed_2,
                           Motor_Spining_Speedy_3 => "DB_Digital_Output".Spin_Carousel_Frequency_Inverter_Speed_3);
END_REGION

REGION Network 7
   RUNG wire#powerrail
      "Instance_FB_Frequency_Inverter_DB_Conveyor_Belt"(Emergency_Stop_Release := "DB_Digital_Input".Emergency_Stop_Release, Start := "DB_Info_From_PCL_Centralizer".Start, Manual_Turn_On_Motor := "DB_Info_From_PCL_Centralizer".Manual_Turn_On_Motor_Conveyor_Belt, Pause_Conveyor_Belt_And_Carousel_Functional_Test := "DB_Contron_Coveyor_Belt".Pause_Conveyor_Belt_And_Carousel_Functional_Test, Select_Motor_Speedy := "DB_Info_From_PCL_Centralizer".Select_Motor_Speed, Motor_Spining_Speedy_1 => "DB_Digital_Output".Conveyor_Belt_Frequency_Inverter_Speed_1, Motor_Spining_Speedy_2 => "DB_Digital_Output".Conveyor_Belt_Frequency_Inverter_Speed_2, Motor_Spining_Speedy_3 => "DB_Digital_Output".Conveyor_Belt_Frequency_Inverter_Speed_3)
   END_RUNG
   // the same network as SCL:
   "Instance_FB_Frequency_Inverter_DB_Conveyor_Belt"(Emergency_Stop_Release := "DB_Digital_Input".Emergency_Stop_Release,   // "FB_Frequency_Inverter"
                           Start := "DB_Info_From_PCL_Centralizer".Start,
                           Manual_Turn_On_Motor := "DB_Info_From_PCL_Centralizer".Manual_Turn_On_Motor_Conveyor_Belt,
                           Pause_Conveyor_Belt_And_Carousel_Functional_Test := "DB_Contron_Coveyor_Belt".Pause_Conveyor_Belt_And_Carousel_Functional_Test,
                           Select_Motor_Speedy := "DB_Info_From_PCL_Centralizer".Select_Motor_Speed,
                           Motor_Spining_Speedy_1 => "DB_Digital_Output".Conveyor_Belt_Frequency_Inverter_Speed_1,
                           Motor_Spining_Speedy_2 => "DB_Digital_Output".Conveyor_Belt_Frequency_Inverter_Speed_2,
                           Motor_Spining_Speedy_3 => "DB_Digital_Output".Conveyor_Belt_Frequency_Inverter_Speed_3);
END_REGION

REGION Network 8
   RUNG wire#powerrail
      "Instance_FB_Send_Water_Fountain_To_Rework_DB"(Emergency_Stop_Release := "DB_Digital_Input".Emergency_Stop_Release, Start := "DB_Info_From_PCL_Centralizer".Start, Water_Fountain_Fail_Test := "DB_Info_From_PCL_Centralizer".Water_Foutain_Fail_Functional_Test, Trigger_Read_Serial_Number_Exit_Functional_Test := "DB_Digital_Input".Sensor_Water_Fountain_Exit_Functional_Test_After_Spinner_Conveyor_Belt, Sensor_Water_Fountain_Exit_Functional_Test_Spinner_Conveyor_Belt := "DB_Digital_Input".Sensor_Water_Fountain_Geting_Entrace_Rework_Conveyor_Belt_Start, Sensor_Spinner_Exit_Functional_Test_Position_Withdrawn := "DB_Digital_Input".Sensor_Water_Fountain_Geting_Entrace_Rework_Conveyor_Belt_Finish, Sensor_Spinner_Exit_Functional_Test_Position_Advanced := "DB_Digital_Input".Carousel_Frequency_Inverter_Fail, Sensor_Water_Fountain_Exit_Functional_Test_After_Spinner_Conveyor_Belt := "DB_Digital_Input".Conveyor_Belt_Functional_Test_Inverter_Fail, Sensor_Water_Fountain_Geting_Entrace_Rework_Conveyor_Belt_Start := "DB_Digital_Input".Selected_Voltage_220V, Turn_On_Conveyor_Belt_Motor_Spinner_Get_Exit_Functional_Test => "DB_Digital_Output".Turn_On_Conveyor_Belt_Motor_Spinner_Get_Exit_Functional_Test, Valve_Advance_Spinner_Get_Exit_Functional_Test => "DB_Digital_Output".Valve_Advance_Spinner_Exit_Functional_Test, Pause_Conveyor_Belt_And_Carousel_Functional_Test => "DB_Contron_Coveyor_Belt".Pause_Conveyor_Belt_And_Carousel_Functional_Test)
   END_RUNG
   // the same network as SCL:
   "Instance_FB_Send_Water_Fountain_To_Rework_DB"(Emergency_Stop_Release := "DB_Digital_Input".Emergency_Stop_Release,   // "FB_Send_Water_Fountain_To_Rework"
                           Start := "DB_Info_From_PCL_Centralizer".Start,
                           Water_Fountain_Fail_Test := "DB_Info_From_PCL_Centralizer".Water_Foutain_Fail_Functional_Test,
                           Trigger_Read_Serial_Number_Exit_Functional_Test := "DB_Digital_Input".Sensor_Water_Fountain_Exit_Functional_Test_After_Spinner_Conveyor_Belt,
                           Sensor_Water_Fountain_Exit_Functional_Test_Spinner_Conveyor_Belt := "DB_Digital_Input".Sensor_Water_Fountain_Geting_Entrace_Rework_Conveyor_Belt_Start,
                           Sensor_Spinner_Exit_Functional_Test_Position_Withdrawn := "DB_Digital_Input".Sensor_Water_Fountain_Geting_Entrace_Rework_Conveyor_Belt_Finish,
                           Sensor_Spinner_Exit_Functional_Test_Position_Advanced := "DB_Digital_Input".Carousel_Frequency_Inverter_Fail,
                           Sensor_Water_Fountain_Exit_Functional_Test_After_Spinner_Conveyor_Belt := "DB_Digital_Input".Conveyor_Belt_Functional_Test_Inverter_Fail,
                           Sensor_Water_Fountain_Geting_Entrace_Rework_Conveyor_Belt_Start := "DB_Digital_Input".Selected_Voltage_220V,
                           Turn_On_Conveyor_Belt_Motor_Spinner_Get_Exit_Functional_Test => "DB_Digital_Output".Turn_On_Conveyor_Belt_Motor_Spinner_Get_Exit_Functional_Test,
                           Valve_Advance_Spinner_Get_Exit_Functional_Test => "DB_Digital_Output".Valve_Advance_Spinner_Exit_Functional_Test,
                           Pause_Conveyor_Belt_And_Carousel_Functional_Test => "DB_Contron_Coveyor_Belt".Pause_Conveyor_Belt_And_Carousel_Functional_Test);
END_REGION

REGION Network 9
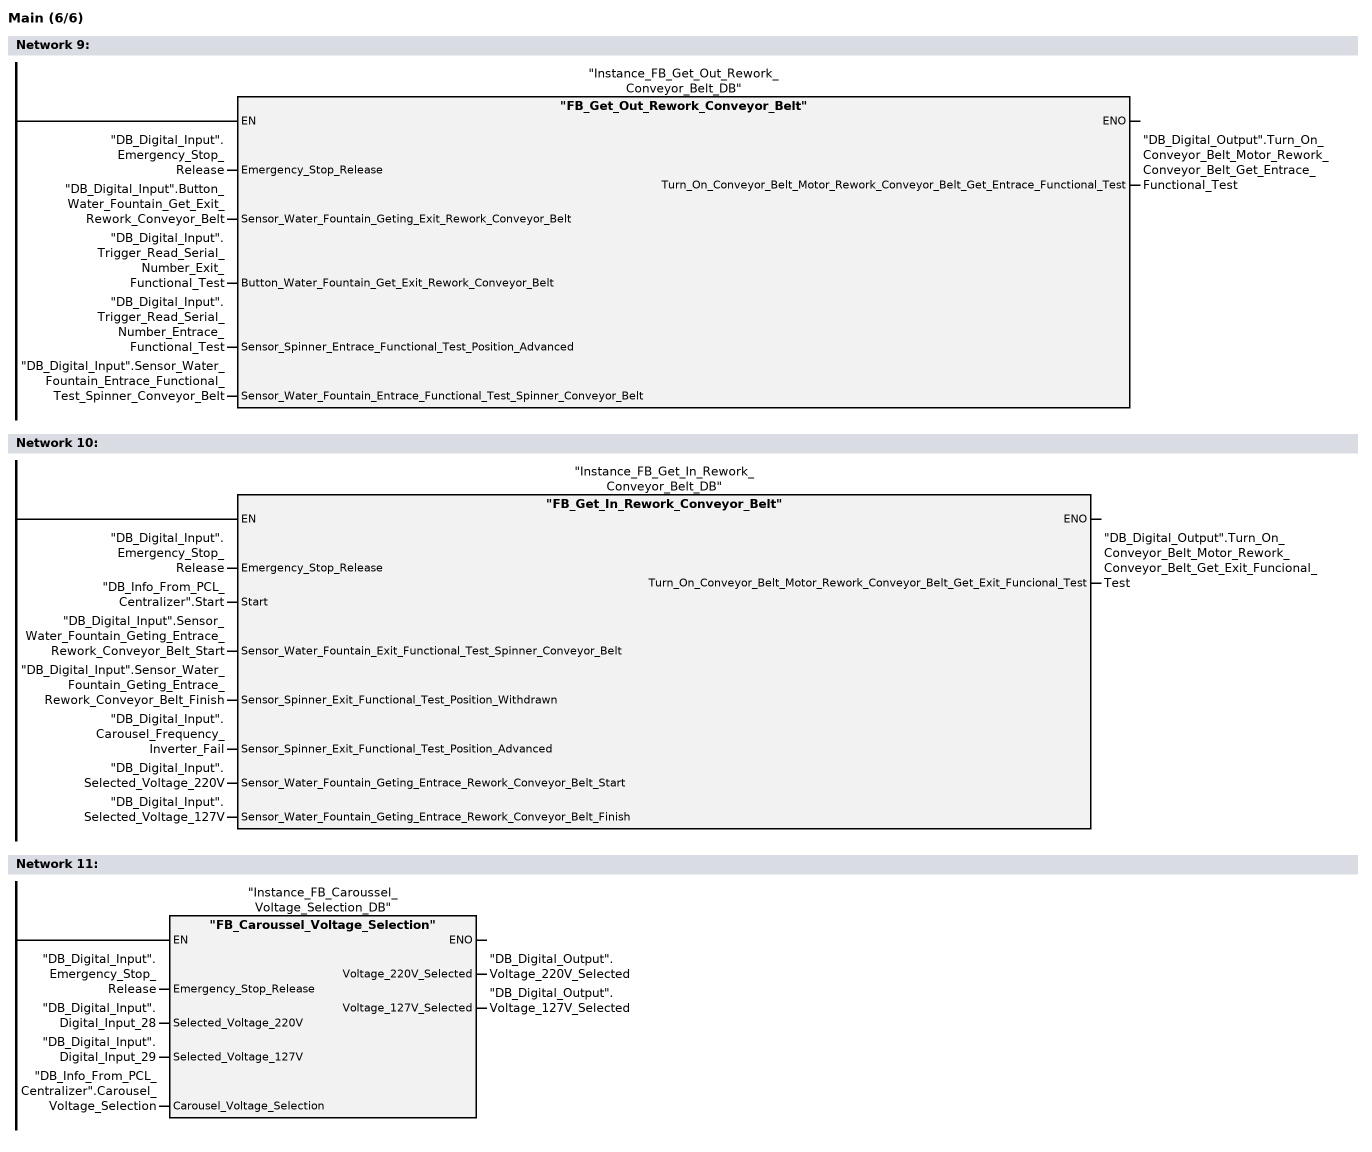
   RUNG wire#powerrail
      "Instance_FB_Get_Out_Rework_Conveyor_Belt_DB"(Emergency_Stop_Release := "DB_Digital_Input".Emergency_Stop_Release, Sensor_Water_Fountain_Geting_Exit_Rework_Conveyor_Belt := "DB_Digital_Input".Button_Water_Fountain_Get_Exit_Rework_Conveyor_Belt, Button_Water_Fountain_Get_Exit_Rework_Conveyor_Belt := "DB_Digital_Input".Trigger_Read_Serial_Number_Exit_Functional_Test, Sensor_Spinner_Entrace_Functional_Test_Position_Advanced := "DB_Digital_Input".Trigger_Read_Serial_Number_Entrace_Functional_Test, Sensor_Water_Fountain_Entrace_Functional_Test_Spinner_Conveyor_Belt := "DB_Digital_Input".Sensor_Water_Fountain_Entrace_Functional_Test_Spinner_Conveyor_Belt, Turn_On_Conveyor_Belt_Motor_Rework_Conveyor_Belt_Get_Entrace_Functional_Test => "DB_Digital_Output".Turn_On_Conveyor_Belt_Motor_Rework_Conveyor_Belt_Get_Entrace_Functional_Test)
   END_RUNG
   // the same network as SCL:
   "Instance_FB_Get_Out_Rework_Conveyor_Belt_DB"(Emergency_Stop_Release := "DB_Digital_Input".Emergency_Stop_Release,   // "FB_Get_Out_Rework_Conveyor_Belt"
                           Sensor_Water_Fountain_Geting_Exit_Rework_Conveyor_Belt := "DB_Digital_Input".Button_Water_Fountain_Get_Exit_Rework_Conveyor_Belt,
                           Button_Water_Fountain_Get_Exit_Rework_Conveyor_Belt := "DB_Digital_Input".Trigger_Read_Serial_Number_Exit_Functional_Test,
                           Sensor_Spinner_Entrace_Functional_Test_Position_Advanced := "DB_Digital_Input".Trigger_Read_Serial_Number_Entrace_Functional_Test,
                           Sensor_Water_Fountain_Entrace_Functional_Test_Spinner_Conveyor_Belt := "DB_Digital_Input".Sensor_Water_Fountain_Entrace_Functional_Test_Spinner_Conveyor_Belt,
                           Turn_On_Conveyor_Belt_Motor_Rework_Conveyor_Belt_Get_Entrace_Functional_Test => "DB_Digital_Output".Turn_On_Conveyor_Belt_Motor_Rework_Conveyor_Belt_Get_Entrace_Functional_Test);
END_REGION

REGION Network 10
   RUNG wire#powerrail
      "Instance_FB_Get_In_Rework_Conveyor_Belt_DB"(Emergency_Stop_Release := "DB_Digital_Input".Emergency_Stop_Release, Start := "DB_Info_From_PCL_Centralizer".Start, Sensor_Water_Fountain_Exit_Functional_Test_Spinner_Conveyor_Belt := "DB_Digital_Input".Sensor_Water_Fountain_Geting_Entrace_Rework_Conveyor_Belt_Start, Sensor_Spinner_Exit_Functional_Test_Position_Withdrawn := "DB_Digital_Input".Sensor_Water_Fountain_Geting_Entrace_Rework_Conveyor_Belt_Finish, Sensor_Spinner_Exit_Functional_Test_Position_Advanced := "DB_Digital_Input".Carousel_Frequency_Inverter_Fail, Sensor_Water_Fountain_Geting_Entrace_Rework_Conveyor_Belt_Start := "DB_Digital_Input".Selected_Voltage_220V, Sensor_Water_Fountain_Geting_Entrace_Rework_Conveyor_Belt_Finish := "DB_Digital_Input".Selected_Voltage_127V, Turn_On_Conveyor_Belt_Motor_Rework_Conveyor_Belt_Get_Exit_Funcional_Test => "DB_Digital_Output".Turn_On_Conveyor_Belt_Motor_Rework_Conveyor_Belt_Get_Exit_Funcional_Test)
   END_RUNG
   // the same network as SCL:
   "Instance_FB_Get_In_Rework_Conveyor_Belt_DB"(Emergency_Stop_Release := "DB_Digital_Input".Emergency_Stop_Release,   // "FB_Get_In_Rework_Conveyor_Belt"
                           Start := "DB_Info_From_PCL_Centralizer".Start,
                           Sensor_Water_Fountain_Exit_Functional_Test_Spinner_Conveyor_Belt := "DB_Digital_Input".Sensor_Water_Fountain_Geting_Entrace_Rework_Conveyor_Belt_Start,
                           Sensor_Spinner_Exit_Functional_Test_Position_Withdrawn := "DB_Digital_Input".Sensor_Water_Fountain_Geting_Entrace_Rework_Conveyor_Belt_Finish,
                           Sensor_Spinner_Exit_Functional_Test_Position_Advanced := "DB_Digital_Input".Carousel_Frequency_Inverter_Fail,
                           Sensor_Water_Fountain_Geting_Entrace_Rework_Conveyor_Belt_Start := "DB_Digital_Input".Selected_Voltage_220V,
                           Sensor_Water_Fountain_Geting_Entrace_Rework_Conveyor_Belt_Finish := "DB_Digital_Input".Selected_Voltage_127V,
                           Turn_On_Conveyor_Belt_Motor_Rework_Conveyor_Belt_Get_Exit_Funcional_Test => "DB_Digital_Output".Turn_On_Conveyor_Belt_Motor_Rework_Conveyor_Belt_Get_Exit_Funcional_Test);
END_REGION

REGION Network 11
   RUNG wire#powerrail
      "Instance_FB_Caroussel_Voltage_Selection_DB"(Emergency_Stop_Release := "DB_Digital_Input".Emergency_Stop_Release, Selected_Voltage_220V := "DB_Digital_Input".Digital_Input_28, Selected_Voltage_127V := "DB_Digital_Input".Digital_Input_29, Carousel_Voltage_Selection := "DB_Info_From_PCL_Centralizer".Carousel_Voltage_Selection, Voltage_220V_Selected => "DB_Digital_Output".Voltage_220V_Selected, Voltage_127V_Selected => "DB_Digital_Output".Voltage_127V_Selected)
   END_RUNG
   // the same network as SCL:
   "Instance_FB_Caroussel_Voltage_Selection_DB"(Emergency_Stop_Release := "DB_Digital_Input".Emergency_Stop_Release,   // "FB_Caroussel_Voltage_Selection"
                           Selected_Voltage_220V := "DB_Digital_Input".Digital_Input_28,
                           Selected_Voltage_127V := "DB_Digital_Input".Digital_Input_29,
                           Carousel_Voltage_Selection := "DB_Info_From_PCL_Centralizer".Carousel_Voltage_Selection,
                           Voltage_220V_Selected => "DB_Digital_Output".Voltage_220V_Selected,
                           Voltage_127V_Selected => "DB_Digital_Output".Voltage_127V_Selected);
END_REGION
END_ORGANIZATION_BLOCK
